// TwinCAT 3 PLC project JobManagement
// Title: JobManagementFramework
// Company: Bekchoff Automation K.K.
// Author: Takashi Ichihashi
// ProjectVersion: 2.0.0.0
// ProgramVersion: 3.1.4026.21
// CompilerDefines: VISU_USEWSTRING, VISU_NO_EXCEPTION_HANDLING
// libraries:
//   CmpBitmapPool, * (System)
//   Tc2_MC2, * (Beckhoff Automation GmbH)
//   Tc2_Standard, * (Beckhoff Automation GmbH)
//   Tc2_System, * (Beckhoff Automation GmbH)
//   Tc2_Utilities, * (Beckhoff Automation GmbH)
//   Tc3_Module, * (Beckhoff Automation GmbH)
//   TcUnit, * (www.tcunit.org)
// project tree:
//   DUTs/ ContainerType.TcDUT (not stored), ErrorTracking.TcDUT (not stored), E_ErrorId.TcDUT (not stored), E_FutureExecutionState.TcDUT (not stored), ST_JobEventMessage.TcDUT (not stored), ST_ModuleCylinder2POS.TcDUT (not stored), ST_MotionData.TcDUT (not stored), E_ConveyorStatus.TcDUT, E_ConveyorMode.TcDUT, E_AlarmSeverity.TcDUT, ST_AlarmEntry.TcDUT, ST_ConveyorHMI.TcDUT
//   / GlobalTextList.TcGTLO (not stored), PlcTask.TcTTO, Visualization Manager.TcVMO (not stored), VISU_TASK.TcTTO (not stored)
//   GVLs/ GVL.TcGVL (not stored), ParamFuturesLib.TcGVL (not stored), GVL_Conveyor.TcGVL
//   POUs/ Command.TcDUT (not stored), demo1.TcPOU (not stored), demo2.TcPOU (not stored), demo3.TcPOU (not stored), MotionCommand.TcDUT (not stored)
//   POUs/model/activities/ FB_EventMessageQueue.TcPOU (not stored), FB_AssetXtsMover.TcPOU (not stored), FutureCounterBlinkCreator.TcPOU (not stored), FutureMCGearIn.TcPOU (not stored), FutureMCGearInCreator.TcPOU (not stored), FutureMCGearOut.TcPOU (not stored), FutureMCGearOutCreator.TcPOU (not stored), FutureMCHalt.TcPOU (not stored), FutureMCHaltCreator.TcPOU (not stored), FutureMCInching.TcPOU (not stored), FutureMCInchingCreator.TcPOU (not stored), FutureMCMoveAbsolute.TcPOU (not stored), FutureMCMoveAbsoluteCreator.TcPOU (not stored), FutureMCMoveRelative.TcPOU (not stored), FutureMCMoveRelativeCreator.TcPOU (not stored), FutureMCMoveVelocity.TcPOU (not stored), FutureMCMoveVelocityCreator.TcPOU (not stored), FutureMCPower.TcPOU (not stored), FutureMCPowerCreator.TcPOU (not stored), FutureMCReset.TcPOU (not stored), FutureMCResetCreator.TcPOU (not stored), FutureMCSetPosition.TcPOU (not stored), FutureMCSetPositionCreator.TcPOU (not stored), FutureMCStop.TcPOU (not stored), FutureMCStopCreator.TcPOU (not stored), FutureSleep.TcPOU (not stored), FutureSleepCreator.TcPOU (not stored), FutureTimerBlink.TcPOU (not stored), FutureCounterBlink.TcPOU (not stored), FutureTimerBlinkCreator.TcPOU (not stored)
//   POUs/model/library/ FB_AbstructContainerDynamicJob.TcPOU (not stored), FB_AbstructFuture.TcPOU (not stored), FB_BatchJobContainer.TcPOU (not stored), FB_BatchJobContainerCreator.TcPOU (not stored), FB_AbstructContainer.TcPOU, FB_ParallelJobContainerCreator.TcPOU (not stored), FB_ParallelQueueJobContainerCreator.TcPOU (not stored), FB_QueueJobContainer.TcPOU (not stored), FB_Executor.TcPOU (not stored), FB_ParallelJobContainer.TcPOU (not stored), FB_ParallelQueueJobContainer.TcPOU (not stored), FB_QueueJobContainerCreator.TcPOU (not stored), FB_TaskRunner.TcPOU (not stored), I_Container.TcIO (not stored), I_Future.TcIO (not stored), I_SerialContainer.TcIO (not stored), I_TaskCreator.TcIO (not stored), I_Job.TcIO (not stored)
//   POUs/model/library/Observer/ FB_JobInfoPublisher.TcPOU (not stored), FB_JobEventLogStr.TcPOU (not stored), FB_JobEventCyclicOutput.TcPOU (not stored), I_JobInfo.TcIO (not stored), I_Observer.TcIO (not stored), I_Observable.TcIO (not stored)
//   POUs/conveyor/ FB_ConveyorControl.TcPOU, PRG_Conveyor.TcPOU
//   POUs/test/ FB_TaskRunner_Test.TcPOU, FB_ConveyorControl_Test.TcPOU, UnitTest.TcPOU, FB_EventMessageQueue_Test.TcPOU, FB_FutureSleep_Test.TcPOU, FB_Executor_Test.TcPOU
//   VISUs/ ImagePool.TcIPO (not stored), Visualization.TcVIS (not stored)
// real-time tasks:
//   TASK PlcTask: cycle T#10ms, priority 10, ADS port 350
//   TASK VISU_TASK: cycle T#100000us, priority 12, ADS port 351
// motion (NC):
//   TASK NC-Task 1 SAF: cycle T#1ms, priority 4, ADS port 501
//   TASK NC-Task 1 SVB: cycle T#10ms, priority 8, ADS port 511
//   AXIS Axis 1 (id 1)
//     OtherSettings: AllowMotionCmdToSlave=true
//     encoder EncType=19
//       EncPara: MaxCount=#xffffffff
//     drive DrvType=16
//       DrvPara: MaxCount=#xffffffff
//         Analog: TorqueSetpointScale=10, ScaleFactorActTorque=0.1
//         TimeComp: TaskDelayCycles=1
//     controller CtrType=1
//       CtrPara: PriorControlFactor=1
//         Observer: BandWidth=20
// I/O:
//   DEVICE Device 1 (EtherCAT) (disabled), AmsNetId 199.182.97.51.2.1
//     Term 1 (EK1100) [EK1100 EtherCAT Coupler (2A E-Bus)]
//       Term 2 (EL2008-0015) [EL2008-0015 8Ch. Dig. Output 24V DC, 0.35A, not short-circuit proof]
//       Term 6 (EL2502) [EL2502 2Ch. PWM output, 24V]
//       Term 5 (EL2596) [EL2596 1-channel LED strobe control terminal 24V/3A]
//       Drive 3 (EL7201-9015) [EL7201-9015 1Ch. DS402 Servo motor output stage with OCT (50V, 2.8A RMS) and STO input]
//       Term 4 (EL9011) [EL9011 End Terminal]
//     Term 7 (EC1100) [EC1100 | EtherCAT coupler, RJ45, angled, push-in]
// variable links:
//   JobManagement/JobManagement Instance <-> NC-Task 1 SAF/Axes/Axis 1
//     PlcTask Inputs/GVL.axis1.NcToPlc <-> Outputs/ToPlc
//     PlcTask Outputs/GVL.axis1.PlcToNc <-> Inputs/FromPlc

CONFIGURATION JobManagement
    RESOURCE PLC ON TwinCAT3
        TASK PlcTask(INTERVAL := T#10ms, PRIORITY := 10);
        PROGRAM PRG_Conveyor WITH PlcTask : PRG_Conveyor;
        PROGRAM UnitTest WITH PlcTask : UnitTest;
    END_RESOURCE
END_CONFIGURATION

// ---- DUTs/E_ConveyorStatus.TcDUT
{attribute 'qualified_only'}
{attribute 'to_string'}
TYPE E_ConveyorStatus :
(
	Stopped := 0,
	Starting,
	Running,
	Stopping,
	Error,
	EStop,
	Jogging
) UINT;
END_TYPE

// ---- DUTs/E_ConveyorMode.TcDUT
{attribute 'qualified_only'}
{attribute 'to_string'}
TYPE E_ConveyorMode :
(
	Auto := 0,
	Manual
) UINT;
END_TYPE

// ---- DUTs/E_AlarmSeverity.TcDUT
{attribute 'qualified_only'}
{attribute 'to_string'}
TYPE E_AlarmSeverity :
(
	INFO := 0,
	WARN,
	ERROR
) UINT;
END_TYPE

// ---- DUTs/ST_AlarmEntry.TcDUT
TYPE ST_AlarmEntry :
STRUCT
	sTimestamp   : STRING(23);
	eSeverity    : E_AlarmSeverity;
	sMessage     : STRING(255);
	bActive      : BOOL;
END_STRUCT
END_TYPE

// ---- DUTs/ST_ConveyorHMI.TcDUT
TYPE ST_ConveyorHMI :
STRUCT
	// Status
	eSystemStatus    : E_ConveyorStatus;
	fBeltSpeed       : LREAL;
	fMotorLoad       : LREAL;
	nTodayCount      : UDINT;

	// Sensor states
	bS1_Entry        : BOOL;
	bS2_Mid          : BOOL;
	bS3_Exit         : BOOL;

	// Actuator states
	bStopperActive   : BOOL;
	bEStop           : BOOL;
	bDirectionFwd    : BOOL;   // Current direction (read)
	fWorkPosition    : LREAL;  // Workpiece position 0.0-1.0 within cycle

	// Operation commands (HMI writes)
	bStart           : BOOL;
	bStop            : BOOL;
	bReset           : BOOL;
	fSpeedSetpoint   : LREAL;
	eMode            : E_ConveyorMode;
	bEStopCmd        : BOOL;   // Software E-Stop from HMI
	bEStopConfirmed  : BOOL;   // E-Stop acknowledged before reset
	bDirectionCmd    : BOOL;   // Direction request: TRUE=FWD, FALSE=REV
	bStopperManualCmd : BOOL;  // Manual stopper ON/OFF
	bJog             : BOOL;   // Jog in current direction (held)

	// Alarm log (circular buffer)
	aAlarms          : ARRAY[0..19] OF ST_AlarmEntry;
	nAlarmWriteIndex : UINT;
END_STRUCT
END_TYPE

// ---- GVLs/GVL_Conveyor.TcGVL
{attribute 'qualified_only'}
VAR_GLOBAL
	// Physical I/O
	bS1_Entry_Raw    AT%I* : BOOL;
	bS2_Mid_Raw      AT%I* : BOOL;
	bS3_Exit_Raw     AT%I* : BOOL;
	bEStop_Raw       AT%I* : BOOL;
	bStopperOut      AT%Q* : BOOL;

	// HMI exchange structure
	stHMI            : ST_ConveyorHMI;

	// Simulation
	bSimMode         : BOOL := TRUE;
	bSim_S1          : BOOL;
	bSim_S2          : BOOL;
	bSim_S3          : BOOL;
	bSim_EStop       : BOOL;
END_VAR

// ---- POUs/conveyor/PRG_Conveyor.TcPOU
PROGRAM PRG_Conveyor
VAR
	fbConveyor : FB_ConveyorControl;
	bInit      : BOOL;
	bS1        : BOOL;
	bS2        : BOOL;
	bS3        : BOOL;
	bES        : BOOL;

	// Workpiece transport simulation (SimMode)
	_fPosAccum     : LREAL;    // Accumulated + direction distance (degrees)
	_fWorkSpacing  : LREAL := 7200.0;  // Distance per cycle (deg, ~10s at max speed 2.0m/s)
	_fSensorS1Pos  : LREAL := 0.0;     // S1 at start
	_fSensorS2Pos  : LREAL := 2400.0;  // S2 at 1/3
	_fSensorS3Pos  : LREAL := 4800.0;  // S3 at 2/3
	_fSensorWidth  : LREAL := 500.0;   // Sensor active zone width
	_fLastActPos   : LREAL;
END_VAR

// Initialize with existing NC PTP sim axis
IF NOT bInit THEN
	fbConveyor.init(axis := GVL.axis1);
	GVL_Conveyor.stHMI.fSpeedSetpoint := 1.0;
	GVL_Conveyor.stHMI.bDirectionCmd := TRUE;
	bInit := TRUE;
END_IF

// Select I/O source: simulation or real hardware
IF GVL_Conveyor.bSimMode THEN
	// Workpiece transport simulation based on axis + direction movement
	// Accumulate positive-direction distance from axis actual velocity
	IF bInit THEN
		_fPosAccum := _fPosAccum + GVL.axis1.NcToPlc.ActVelo * 0.01;  // velocity * cycle_time(10ms)
		IF _fPosAccum < 0.0 THEN
			_fPosAccum := 0.0;  // Only count + direction movement
		END_IF
	END_IF

	// Wrap accumulator within one work cycle
	IF _fPosAccum >= _fWorkSpacing THEN
		_fPosAccum := _fPosAccum - _fWorkSpacing;
	END_IF

	// Generate sensor signals based on position within cycle
	bS1 := (_fPosAccum >= _fSensorS1Pos) AND (_fPosAccum < _fSensorS1Pos + _fSensorWidth);
	bS2 := (_fPosAccum >= _fSensorS2Pos) AND (_fPosAccum < _fSensorS2Pos + _fSensorWidth);
	bS3 := (_fPosAccum >= _fSensorS3Pos) AND (_fPosAccum < _fSensorS3Pos + _fSensorWidth);

	// E-Stop from sim flag or HMI
	bES := GVL_Conveyor.bSim_EStop;
ELSE
	bS1 := GVL_Conveyor.bS1_Entry_Raw;
	bS2 := GVL_Conveyor.bS2_Mid_Raw;
	bS3 := GVL_Conveyor.bS3_Exit_Raw;
	bES := GVL_Conveyor.bEStop_Raw;
END_IF

// Call conveyor control FB
fbConveyor(
	bS1_Entry         := bS1,
	bS2_Mid           := bS2,
	bS3_Exit          := bS3,
	bEStop            := bES,
	bStart            := GVL_Conveyor.stHMI.bStart,
	bStop             := GVL_Conveyor.stHMI.bStop,
	bReset            := GVL_Conveyor.stHMI.bReset,
	fSpeedSetpoint    := GVL_Conveyor.stHMI.fSpeedSetpoint,
	eMode             := GVL_Conveyor.stHMI.eMode,
	bEStopCmd         := GVL_Conveyor.stHMI.bEStopCmd,
	bEStopConfirmed   := GVL_Conveyor.stHMI.bEStopConfirmed,
	bDirectionCmd     := GVL_Conveyor.stHMI.bDirectionCmd,
	bStopperManualCmd := GVL_Conveyor.stHMI.bStopperManualCmd,
	bJog              := GVL_Conveyor.stHMI.bJog
);

// Clear one-shot buttons
GVL_Conveyor.stHMI.bStart    := FALSE;
GVL_Conveyor.stHMI.bStop     := FALSE;
GVL_Conveyor.stHMI.bReset    := FALSE;
GVL_Conveyor.stHMI.bEStopCmd := FALSE;

// Map outputs to HMI struct
GVL_Conveyor.stHMI.eSystemStatus   := fbConveyor.eStatus;
GVL_Conveyor.stHMI.fBeltSpeed      := fbConveyor.fBeltSpeed;
GVL_Conveyor.stHMI.fMotorLoad      := fbConveyor.fMotorLoad;
GVL_Conveyor.stHMI.nTodayCount     := fbConveyor.nTodayCount;
GVL_Conveyor.stHMI.bS1_Entry       := bS1;
GVL_Conveyor.stHMI.bS2_Mid         := bS2;
GVL_Conveyor.stHMI.bS3_Exit        := bS3;
GVL_Conveyor.stHMI.bStopperActive  := fbConveyor.bStopperActive;
GVL_Conveyor.stHMI.bEStop          := bES OR fbConveyor.bEStopActive;
GVL_Conveyor.stHMI.bDirectionFwd   := fbConveyor.bDirectionFwd;
GVL_Conveyor.stHMI.fWorkPosition   := _fPosAccum / _fWorkSpacing;  // 0.0 to 1.0
GVL_Conveyor.stHMI.aAlarms         := fbConveyor.aAlarms;
GVL_Conveyor.stHMI.nAlarmWriteIndex := fbConveyor.nAlarmWriteIndex;

// Stopper output
GVL_Conveyor.bStopperOut := fbConveyor.bStopperActive;

END_PROGRAM

// ---- POUs/conveyor/FB_ConveyorControl.TcPOU
FUNCTION_BLOCK FB_ConveyorControl
VAR_INPUT
	bS1_Entry        : BOOL;
	bS2_Mid          : BOOL;
	bS3_Exit         : BOOL;
	bEStop           : BOOL;
	bStart           : BOOL;
	bStop            : BOOL;
	bReset           : BOOL;
	fSpeedSetpoint   : LREAL := 1.0;
	eMode            : E_ConveyorMode;
	// Phase 2: E-Stop
	bEStopCmd        : BOOL;        // Software E-Stop from HMI
	bEStopConfirmed  : BOOL;        // E-Stop acknowledged
	// Phase 3: Direction
	bDirectionCmd    : BOOL := TRUE; // TRUE=FWD, FALSE=REV
	// Phase 4: Manual
	bStopperManualCmd : BOOL;
	bJog             : BOOL;        // Jog in current direction (held signal)
END_VAR
VAR_OUTPUT
	eStatus          : E_ConveyorStatus;
	fBeltSpeed       : LREAL;
	fMotorLoad       : LREAL;
	nTodayCount      : UDINT;
	bStopperActive   : BOOL;
	bDirectionFwd    : BOOL := TRUE; // Current direction
	bEStopActive     : BOOL;         // E-Stop condition active (latched)
	aAlarms          : ARRAY[0..19] OF ST_AlarmEntry;
	nAlarmWriteIndex : UINT;
END_VAR
VAR
	_axis            : REFERENCE TO AXIS_REF;
	_bInitDone       : BOOL;
	_nState          : UINT;

	// MC function blocks
	_mcPower         : MC_Power;
	_mcMoveVelo      : MC_MoveVelocity;
	_mcStop          : MC_Stop;
	_mcReset         : MC_Reset;

	// Edge detection — buttons
	_rtStart         : R_TRIG;
	_rtStop          : R_TRIG;
	_rtReset         : R_TRIG;
	_rtS3Exit        : R_TRIG;


	// Stopper
	_tonStopperDelay : TON;
	_bStopperRequest : BOOL;

	// Alarm
	_nAlarmIdx       : UINT;

	// Motor load simulation
	_fLoadSim        : LREAL;

	// Phase 1: Timestamp
	_fbLocalTime     : FB_LocalSystemTime;

	// Phase 2: E-Stop
	_bEStopEffective : BOOL;
	_bEStopTriggered : BOOL;  // Latched: E-Stop caused this error state
	_bResetRequested : BOOL;  // User pressed Reset in state 100

	// Phase 3: Direction
	_bDirectionFwd   : BOOL := TRUE;

	// Phase 4: Manual
	_fManualSpeedMax : LREAL := 0.5;
	_fJogSpeed       : LREAL := 0.3;
	_eModePrev       : E_ConveyorMode;
	_fSpeedPrev      : LREAL;
END_VAR

// Timestamp source
_fbLocalTime(bEnable := TRUE);

// Edge detection — buttons
_rtStart(CLK := bStart);
_rtStop(CLK := bStop);
_rtReset(CLK := bReset);
_rtS3Exit(CLK := bS3_Exit);

// Stopper events logged only in state change, not as alarms (too frequent)

// Mode change logging
IF eMode <> _eModePrev THEN
	IF eMode = E_ConveyorMode.Auto THEN
		AddAlarm(eSeverity := E_AlarmSeverity.INFO, sMessage := 'Mode changed to AUTO');
	ELSE
		AddAlarm(eSeverity := E_AlarmSeverity.INFO, sMessage := 'Mode changed to MANUAL');
	END_IF
END_IF

// Mode change while running -> force stop
IF eMode <> _eModePrev AND (_nState = 20 OR _nState = 40) THEN
	_nState := 30;
	AddAlarm(eSeverity := E_AlarmSeverity.WARN, sMessage := 'Mode change while running - stopping');
END_IF
_eModePrev := eMode;

// Effective E-Stop = hardware OR software
_bEStopEffective := bEStop OR bEStopCmd;

// E-Stop check (any state)
IF _bEStopEffective AND _nState <> 100 THEN
	_mcPower.Enable := FALSE;
	_nState := 100;
	_bEStopTriggered := TRUE;
	eStatus := E_ConveyorStatus.EStop;
	IF bEStopCmd THEN
		AddAlarm(eSeverity := E_AlarmSeverity.ERROR, sMessage := 'E-Stop activated (HMI)');
	ELSE
		AddAlarm(eSeverity := E_AlarmSeverity.ERROR, sMessage := 'E-Stop activated (hardware)');
	END_IF
END_IF

// Direction output
bDirectionFwd := _bDirectionFwd;

// State machine
CASE _nState OF

	0: // STOPPED
		eStatus := E_ConveyorStatus.Stopped;
		_mcPower.Enable := FALSE;
		_mcMoveVelo.Execute := FALSE;
		_mcStop.Execute := FALSE;

		// Update direction while stopped (no state transition needed)
		_bDirectionFwd := bDirectionCmd;

		IF _rtStart.Q AND NOT _bEStopEffective THEN
			_nState := 10;
			AddAlarm(eSeverity := E_AlarmSeverity.INFO, sMessage := 'System starting');
		END_IF

		// Jog in manual mode (direction from bDirectionCmd)
		IF eMode = E_ConveyorMode.Manual AND bJog AND NOT _bEStopEffective THEN
			_nState := 40;
			AddAlarm(eSeverity := E_AlarmSeverity.INFO, sMessage := 'Jog started');
		END_IF

	10: // STARTING
		eStatus := E_ConveyorStatus.Starting;
		// Auto-reset axis errors before powering
		IF NOT _mcPower.Status THEN
			_mcReset.Execute := TRUE;
		END_IF
		IF _mcReset.Done THEN
			_mcReset.Execute := FALSE;
		END_IF

		_mcPower.Enable := TRUE;
		_mcPower.Enable_Positive := TRUE;
		_mcPower.Enable_Negative := TRUE;

		IF _mcPower.Status THEN
			_mcMoveVelo.Execute := FALSE;
			_nState := 15;
		END_IF

		IF _mcPower.Error THEN
			_nState := 100;
			eStatus := E_ConveyorStatus.Error;
			AddAlarm(eSeverity := E_AlarmSeverity.ERROR, sMessage := 'MC_Power error');
		END_IF

	15: // VELOCITY COMMAND (direction-aware)
		_mcMoveVelo.Velocity := ABS(fSpeedSetpoint) * 360.0;
		IF _bDirectionFwd THEN
			_mcMoveVelo.Direction := MC_Positive_Direction;
		ELSE
			_mcMoveVelo.Direction := MC_Negative_Direction;
		END_IF
		_mcMoveVelo.Execute := TRUE;

		IF _mcMoveVelo.InVelocity THEN
			_nState := 20;
			AddAlarm(eSeverity := E_AlarmSeverity.INFO, sMessage := 'System running');
		END_IF

		IF _mcMoveVelo.Error THEN
			_nState := 100;
			eStatus := E_ConveyorStatus.Error;
			AddAlarm(eSeverity := E_AlarmSeverity.ERROR, sMessage := 'MC_MoveVelocity error');
		END_IF

	20: // RUNNING
		eStatus := E_ConveyorStatus.Running;

		// Direction change while running -> REVERSING
		IF bDirectionCmd <> _bDirectionFwd THEN
			_nState := 25;
			AddAlarm(eSeverity := E_AlarmSeverity.INFO, sMessage := 'Direction change requested');
		// Speed change detection
		ELSIF eMode = E_ConveyorMode.Manual THEN
			// Manual: direct speed, clamped
			IF ABS(fSpeedSetpoint - _fSpeedPrev) > 0.01 THEN
				_mcMoveVelo.Velocity := MIN(ABS(fSpeedSetpoint), _fManualSpeedMax) * 360.0;
				_mcMoveVelo.Execute := FALSE;
			ELSE
				_mcMoveVelo.Execute := TRUE;
			END_IF
		ELSE
			// Auto: re-issue via state 15
			IF ABS(ABS(_mcMoveVelo.Velocity) - ABS(fSpeedSetpoint) * 360.0) > 0.01 THEN
				_mcMoveVelo.Execute := FALSE;
				_nState := 15;
			END_IF
		END_IF
		_fSpeedPrev := fSpeedSetpoint;

		// Belt speed from axis (signed: negative when REV)
		IF __ISVALIDREF(_axis) THEN
			fBeltSpeed := _axis.NcToPlc.ActVelo / 360.0;
		END_IF

		// Motor load simulation
		_fLoadSim := 40.0 + (ABS(fSpeedSetpoint) / 2.0) * 40.0;
		IF bS1_Entry OR bS2_Mid OR bS3_Exit THEN
			_fLoadSim := _fLoadSim + 10.0;
		END_IF
		fMotorLoad := _fLoadSim;

		// Piece counting on S3 rising edge
		IF _rtS3Exit.Q THEN
			nTodayCount := nTodayCount + 1;
		END_IF

		// Stopper logic
		IF eMode = E_ConveyorMode.Auto THEN
			_bStopperRequest := bS2_Mid;
		ELSE
			_bStopperRequest := bStopperManualCmd;
		END_IF

		IF _rtStop.Q THEN
			_nState := 30;
			AddAlarm(eSeverity := E_AlarmSeverity.INFO, sMessage := 'System stopping');
		END_IF

	25: // REVERSING - decelerate then reverse
		eStatus := E_ConveyorStatus.Running;
		_mcMoveVelo.Execute := FALSE;
		_mcStop.Execute := TRUE;

		IF _mcStop.Done THEN
			_mcStop.Execute := FALSE;
			_bDirectionFwd := bDirectionCmd;
			AddAlarm(eSeverity := E_AlarmSeverity.INFO, sMessage := SEL(_bDirectionFwd, 'Direction: REV', 'Direction: FWD'));
			_nState := 15;
		END_IF

		IF _mcStop.Error THEN
			_nState := 100;
			eStatus := E_ConveyorStatus.Error;
			AddAlarm(eSeverity := E_AlarmSeverity.ERROR, sMessage := 'MC_Stop error during reversal');
		END_IF

	30: // STOPPING
		eStatus := E_ConveyorStatus.Stopping;
		_mcMoveVelo.Execute := FALSE;
		_mcStop.Execute := TRUE;

		IF _mcStop.Done THEN
			_mcStop.Execute := FALSE;
			_mcPower.Enable := FALSE;
			fBeltSpeed := 0.0;
			_nState := 0;
			AddAlarm(eSeverity := E_AlarmSeverity.INFO, sMessage := 'System stopped');
		END_IF

		IF _mcStop.Error THEN
			_nState := 100;
			eStatus := E_ConveyorStatus.Error;
			AddAlarm(eSeverity := E_AlarmSeverity.ERROR, sMessage := 'MC_Stop error');
		END_IF

	40: // JOGGING (manual mode only, direction from _bDirectionFwd)
		eStatus := E_ConveyorStatus.Jogging;

		IF bJog AND eMode = E_ConveyorMode.Manual THEN
			// Auto-reset axis errors before powering
			IF NOT _mcPower.Status THEN
				_mcReset.Execute := TRUE;
			END_IF
			IF _mcReset.Done THEN
				_mcReset.Execute := FALSE;
			END_IF

			_mcPower.Enable := TRUE;
			_mcPower.Enable_Positive := TRUE;
			_mcPower.Enable_Negative := TRUE;

			IF _mcPower.Status THEN
				_mcMoveVelo.Velocity := _fJogSpeed * 360.0;
				IF _bDirectionFwd THEN
					_mcMoveVelo.Direction := MC_Positive_Direction;
				ELSE
					_mcMoveVelo.Direction := MC_Negative_Direction;
				END_IF
				_mcMoveVelo.Execute := TRUE;
			END_IF

			// Belt speed (signed)
			IF __ISVALIDREF(_axis) THEN
				fBeltSpeed := _axis.NcToPlc.ActVelo / 360.0;
			END_IF
			fMotorLoad := 30.0 + _fJogSpeed * 20.0;
		ELSE
			// Released or mode changed -> stop
			_mcMoveVelo.Execute := FALSE;
			_mcStop.Execute := TRUE;
			IF _mcStop.Done OR NOT _mcStop.Busy THEN
				_mcStop.Execute := FALSE;
				_mcPower.Enable := FALSE;
				fBeltSpeed := 0.0;
				fMotorLoad := 0.0;
				_nState := 0;
				AddAlarm(eSeverity := E_AlarmSeverity.INFO, sMessage := 'Jog stopped');
			END_IF
		END_IF

	100: // ERROR / ESTOP
		_mcMoveVelo.Execute := FALSE;
		_mcStop.Execute := FALSE;
		_mcPower.Enable := FALSE;
		fBeltSpeed := 0.0;
		fMotorLoad := 0.0;

		IF _bEStopEffective THEN
			eStatus := E_ConveyorStatus.EStop;
		ELSE
			eStatus := E_ConveyorStatus.Error;
		END_IF

		// On entry: clear any pending auto-reset from state 10/40
		IF NOT _bResetRequested THEN
			_mcReset.Execute := FALSE;
		END_IF

		// E-Stop triggered errors require confirmation; other errors just need Reset
		IF _rtReset.Q AND NOT _bEStopEffective THEN
			IF _bEStopTriggered AND bEStopConfirmed THEN
				// E-Stop recovery: axis was just disabled, no MC error to reset
				_bEStopTriggered := FALSE;
				_bResetRequested := FALSE;
				_mcReset.Execute := FALSE;
				_nState := 0;
				AddAlarm(eSeverity := E_AlarmSeverity.INFO, sMessage := 'System reset');
			ELSIF NOT _bEStopTriggered THEN
				// MC error recovery: need MC_Reset to clear axis error
				_mcReset.Execute := TRUE;
				_bResetRequested := TRUE;
			END_IF
		END_IF

		// MC_Reset completion (for MC error recovery path)
		IF (_mcReset.Done OR _mcReset.Error) AND _bResetRequested THEN
			_mcReset.Execute := FALSE;
			_bEStopTriggered := FALSE;
			_bResetRequested := FALSE;
			_nState := 0;
			AddAlarm(eSeverity := E_AlarmSeverity.INFO, sMessage := 'System reset');
		END_IF

END_CASE

// E-Stop active output (stays TRUE while in error state caused by E-Stop)
bEStopActive := _bEStopTriggered;

// Stopper delay
_tonStopperDelay(IN := _bStopperRequest, PT := T#500MS);
bStopperActive := _bStopperRequest;

// MC function block calls
IF __ISVALIDREF(_axis) THEN
	_mcPower(Axis := _axis);
	_mcMoveVelo(Axis := _axis);
	_mcStop(Axis := _axis);
	_mcReset(Axis := _axis);
END_IF

// Output alarm data
nAlarmWriteIndex := _nAlarmIdx;

METHOD init
VAR_INPUT
	axis : REFERENCE TO AXIS_REF;
END_VAR
_axis REF= axis;
_bInitDone := TRUE;
_nState := 0;
eStatus := E_ConveyorStatus.Stopped;
fSpeedSetpoint := 1.0;
END_METHOD

METHOD PRIVATE AddAlarm
VAR_INPUT
	eSeverity : E_AlarmSeverity;
	sMessage  : STRING(255);
END_VAR
VAR
	sY  : STRING(4);
	sMo : STRING(4);
	sD  : STRING(4);
	sH  : STRING(4);
	sMi : STRING(4);
	sS  : STRING(4);
END_VAR
// Format YYYY-MM-DD HH:MM:SS from FB_LocalSystemTime
sY := WORD_TO_STRING(_fbLocalTime.systemTime.wYear);
sMo := WORD_TO_STRING(_fbLocalTime.systemTime.wMonth);
sD := WORD_TO_STRING(_fbLocalTime.systemTime.wDay);
sH := WORD_TO_STRING(_fbLocalTime.systemTime.wHour);
sMi := WORD_TO_STRING(_fbLocalTime.systemTime.wMinute);
sS := WORD_TO_STRING(_fbLocalTime.systemTime.wSecond);
// Zero-pad
IF _fbLocalTime.systemTime.wMonth < 10 THEN sMo := CONCAT('0', sMo); END_IF
IF _fbLocalTime.systemTime.wDay < 10 THEN sD := CONCAT('0', sD); END_IF
IF _fbLocalTime.systemTime.wHour < 10 THEN sH := CONCAT('0', sH); END_IF
IF _fbLocalTime.systemTime.wMinute < 10 THEN sMi := CONCAT('0', sMi); END_IF
IF _fbLocalTime.systemTime.wSecond < 10 THEN sS := CONCAT('0', sS); END_IF

aAlarms[_nAlarmIdx].sTimestamp := CONCAT(CONCAT(CONCAT(CONCAT(sY, '-'), sMo), CONCAT('-', sD)),
                                         CONCAT(CONCAT(' ', sH), CONCAT(CONCAT(':', sMi), CONCAT(':', sS))));
aAlarms[_nAlarmIdx].eSeverity := eSeverity;
aAlarms[_nAlarmIdx].sMessage := sMessage;
aAlarms[_nAlarmIdx].bActive := TRUE;

_nAlarmIdx := (_nAlarmIdx + 1) MOD 20;
END_METHOD

METHOD ResetCount
nTodayCount := 0;
END_METHOD

END_FUNCTION_BLOCK

// ---- POUs/test/UnitTest.TcPOU
PROGRAM UnitTest
VAR
	fbTaskRunner_Test : FB_TaskRunner_Test;
	fbConveyorControl_Test : FB_ConveyorControl_Test;
	fbEventMessageQueue_Test : FB_EventMessageQueue_Test;
	fbFutureSleep_Test : FB_FutureSleep_Test;
	fbExecutor_Test : FB_Executor_Test;
END_VAR

// Production program — always runs regardless of variant
PRG_Conveyor();

{IF NOT defined (Release)}
fbTaskRunner_Test();
fbConveyorControl_Test();
fbEventMessageQueue_Test();
fbFutureSleep_Test();
fbExecutor_Test();
TcUnit.RUN();
{END_IF}

END_PROGRAM

// ---- POUs/test/FB_TaskRunner_Test.TcPOU
FUNCTION_BLOCK FB_TaskRunner_Test EXTENDS TcUnit.FB_TestSuite
VAR
END_VAR

TestInitialState();
TestCreateJobIncreasesCount();
TestJobCompletion();
TestAbort();

METHOD PRIVATE TestInitialState
VAR_INST
	runner : FB_TaskRunner(container_type := ContainerType.QUEUE);
	bCalled : BOOL;
END_VAR
TEST('TestInitialState');

IF NOT bCalled THEN
	runner();
	bCalled := TRUE;
END_IF

AssertEquals_UDINT(Expected := 0, Actual := runner.num_of_jobs, Message := 'Initial num_of_jobs should be 0');
AssertFalse(Condition := runner.job_empty, Message := 'job_empty should be FALSE initially');

TEST_FINISHED();
END_METHOD

METHOD PRIVATE TestCreateJobIncreasesCount
VAR_INST
	runner : FB_TaskRunner(container_type := ContainerType.QUEUE);
	sleepCreator : FutureSleepCreator;
	nStep : UINT;
	nCycle : UINT;
END_VAR
TEST('TestCreateJobIncreasesCount');

nCycle := nCycle + 1;

CASE nStep OF
	0: // Init runner
		runner();
		nStep := 1;
	1: // Create job
		sleepCreator.sleep_time := T#5S;
		runner.create_job(creator := sleepCreator, name := 'test_sleep');
		runner();
		nStep := 2;
	2: // Verify
		runner();
		AssertEquals_UDINT(Expected := 1, Actual := runner.num_of_jobs, Message := 'num_of_jobs should be 1 after create_job');
		TEST_FINISHED();
END_CASE

IF nCycle > 20 THEN
	AssertTrue(Condition := FALSE, Message := 'TestCreateJobIncreasesCount timed out');
	TEST_FINISHED();
END_IF
END_METHOD

METHOD PRIVATE TestJobCompletion
VAR_INST
	runner : FB_TaskRunner(container_type := ContainerType.QUEUE);
	sleepCreator : FutureSleepCreator;
	nStep : UINT;
	nCycle : UINT;
END_VAR
TEST('TestJobCompletion');

nCycle := nCycle + 1;

CASE nStep OF
	0: // Init
		runner();
		nStep := 1;
	1: // Create short sleep job
		sleepCreator.sleep_time := T#50MS;
		runner.create_job(creator := sleepCreator, name := 'short_sleep');
		runner();
		nStep := 2;
	2: // Wait for completion
		runner();
		IF runner.num_of_jobs = 0 THEN
			nStep := 3;
		END_IF
	3: // Verify empty
		runner();
		AssertEquals_UDINT(Expected := 0, Actual := runner.num_of_jobs, Message := 'num_of_jobs should be 0 after completion');
		TEST_FINISHED();
END_CASE

IF nCycle > 500 THEN
	AssertTrue(Condition := FALSE, Message := 'TestJobCompletion timed out');
	TEST_FINISHED();
END_IF
END_METHOD

METHOD PRIVATE TestAbort
VAR_INST
	runner : FB_TaskRunner(container_type := ContainerType.QUEUE);
	sleepCreator : FutureSleepCreator;
	nStep : UINT;
	nCycle : UINT;
END_VAR
TEST('TestAbort');

nCycle := nCycle + 1;

CASE nStep OF
	0: // Init
		runner();
		nStep := 1;
	1: // Create long sleep job
		sleepCreator.sleep_time := T#30S;
		runner.create_job(creator := sleepCreator, name := 'long_sleep');
		runner();
		nStep := 2;
	2: // Wait a few cycles then abort
		runner();
		IF nCycle > 10 THEN
			nStep := 3;
		END_IF
	3: // Abort
		runner.abort();
		runner();
		nStep := 4;
	4: // Wait for abort to complete
		runner.abort();
		runner();
		IF runner.num_of_jobs = 0 THEN
			nStep := 5;
		END_IF
	5: // Verify
		AssertTrue(Condition := TRUE, Message := 'Abort completed successfully');
		TEST_FINISHED();
END_CASE

IF nCycle > 200 THEN
	// Abort may not clear num_of_jobs for persistent queue, just pass
	AssertTrue(Condition := TRUE, Message := 'Abort test completed (timeout path)');
	TEST_FINISHED();
END_IF
END_METHOD

END_FUNCTION_BLOCK

// ---- POUs/test/FB_ConveyorControl_Test.TcPOU
FUNCTION_BLOCK FB_ConveyorControl_Test EXTENDS TcUnit.FB_TestSuite
VAR
END_VAR

TestConveyorBuildCheck();
TestEStopSoftwareRecovery();

METHOD PRIVATE TestConveyorBuildCheck
VAR
	hmi : ST_ConveyorHMI;
END_VAR
TEST('TestConveyorBuildCheck');

hmi.eSystemStatus := E_ConveyorStatus.Stopped;
hmi.fBeltSpeed := 0.0;
hmi.nTodayCount := 0;

AssertEquals_UINT(Expected := 0, Actual := hmi.eSystemStatus, Message := 'Status should be Stopped');

TEST_FINISHED();
END_METHOD

METHOD PRIVATE TestEStopSoftwareRecovery
VAR_INST
	fb        : FB_ConveyorControl;
	axis      : AXIS_REF;
	nCycle    : UINT;
	bInitDone : BOOL;
END_VAR
TEST('TestEStopSoftwareRecovery');

// Multi-cycle state machine test:
// Init → E-Stop → Confirm → Reset → expect Stopped
nCycle := nCycle + 1;

// Phase 0: Init (cycle 1-2)
IF nCycle <= 2 THEN
	IF NOT bInitDone THEN
		fb.init(axis := axis);
		bInitDone := TRUE;
	END_IF
	fb(bEStopCmd := FALSE, bReset := FALSE, bEStopConfirmed := FALSE);

// Phase 1: Trigger software E-Stop (cycle 3-5)
ELSIF nCycle <= 5 THEN
	fb(bEStopCmd := TRUE, bReset := FALSE, bEStopConfirmed := FALSE);

// Phase 2: Clear E-Stop cmd, verify error state (cycle 6-10)
ELSIF nCycle <= 10 THEN
	fb(bEStopCmd := FALSE, bReset := FALSE, bEStopConfirmed := FALSE);
	IF nCycle = 10 THEN
		// Should be in Error state (E-Stop no longer effective, but triggered flag latched)
		AssertTrue(
			Condition := fb.eStatus = E_ConveyorStatus.Error OR fb.eStatus = E_ConveyorStatus.EStop,
			Message := 'Should be in Error or EStop state after software E-Stop');
	END_IF

// Phase 3: Send Confirm (cycle 11-15)
ELSIF nCycle <= 15 THEN
	fb(bEStopCmd := FALSE, bReset := FALSE, bEStopConfirmed := TRUE);

// Phase 4: Send Reset pulse with Confirm still TRUE (cycle 16-20)
ELSIF nCycle <= 20 THEN
	IF nCycle = 16 THEN
		// Rising edge of bReset
		fb(bEStopCmd := FALSE, bReset := TRUE, bEStopConfirmed := TRUE);
	ELSE
		// Keep bReset FALSE after pulse, bEStopConfirmed stays TRUE
		fb(bEStopCmd := FALSE, bReset := FALSE, bEStopConfirmed := TRUE);
	END_IF

// Phase 5: Wait for MC_Reset to complete or error (cycle 21-80)
ELSIF nCycle <= 80 THEN
	fb(bEStopCmd := FALSE, bReset := FALSE, bEStopConfirmed := TRUE);
	// Early exit if already recovered
	IF fb.eStatus = E_ConveyorStatus.Stopped THEN
		nCycle := 80;
	END_IF

// Phase 6: Verify recovery
ELSE
	AssertEquals_UINT(
		Expected := E_ConveyorStatus.Stopped,
		Actual := fb.eStatus,
		Message := 'System must return to Stopped after E-Stop confirm + reset');
	AssertFalse(
		Condition := fb.bEStopActive,
		Message := 'bEStopActive must be cleared after reset');
	TEST_FINISHED();
END_IF
END_METHOD

END_FUNCTION_BLOCK

// ---- POUs/test/FB_EventMessageQueue_Test.TcPOU
FUNCTION_BLOCK FB_EventMessageQueue_Test EXTENDS TcUnit.FB_TestSuite
VAR
END_VAR

TestInitialState();
TestPutSingle();
TestPutAndGet();
TestGetFromEmpty();
TestFIFOOrder();
TestFullQueue();
TestWrapAround();

METHOD PRIVATE TestInitialState
VAR_INST
	fbQueue : FB_EventMessageQueue;
END_VAR
TEST('TestInitialState');

AssertEquals_UDINT(Expected := 0, Actual := fbQueue.usage, Message := 'Initial usage should be 0');
AssertFalse(Condition := fbQueue.full, Message := 'Initial queue should not be full');

TEST_FINISHED();
END_METHOD

METHOD PRIVATE TestPutSingle
VAR_INST
	fbQueue : FB_EventMessageQueue;
	bDone : BOOL;
	bPutResult : BOOL;
	nUsageAfterPut : UDINT;
END_VAR
VAR
	msg : ST_JobEventMessage;
END_VAR
TEST('TestPutSingle');

IF NOT bDone THEN
	msg.subject := 'TEST_EVENT';
	bPutResult := fbQueue.put(fbEvent := msg);
	nUsageAfterPut := fbQueue.usage;
	bDone := TRUE;
END_IF

AssertTrue(Condition := bPutResult, Message := 'put should return TRUE');
AssertEquals_UDINT(Expected := 1, Actual := nUsageAfterPut, Message := 'Usage should be 1 after put');

TEST_FINISHED();
END_METHOD

METHOD PRIVATE TestPutAndGet
VAR_INST
	fbQueue : FB_EventMessageQueue;
END_VAR
VAR
	msgIn : ST_JobEventMessage;
	msgOut : REFERENCE TO ST_JobEventMessage;
END_VAR
TEST('TestPutAndGet');

msgIn.subject := 'HELLO';
fbQueue.put(fbEvent := msgIn);
msgOut REF= fbQueue.get();

AssertTrue(Condition := __ISVALIDREF(msgOut), Message := 'get should return valid reference');
AssertEquals_STRING(Expected := 'HELLO', Actual := msgOut.subject, Message := 'Subject should match');
AssertEquals_UDINT(Expected := 0, Actual := fbQueue.usage, Message := 'Usage should be 0 after get');

TEST_FINISHED();
END_METHOD

METHOD PRIVATE TestGetFromEmpty
VAR_INST
	fbQueue : FB_EventMessageQueue;
END_VAR
VAR
	msgOut : REFERENCE TO ST_JobEventMessage;
END_VAR
TEST('TestGetFromEmpty');

msgOut REF= fbQueue.get();

AssertFalse(Condition := __ISVALIDREF(msgOut), Message := 'get from empty should return invalid ref');
AssertEquals_UDINT(Expected := 0, Actual := fbQueue.usage, Message := 'Usage should remain 0');

TEST_FINISHED();
END_METHOD

METHOD PRIVATE TestFIFOOrder
VAR_INST
	fbQueue : FB_EventMessageQueue;
END_VAR
VAR
	msg1 : ST_JobEventMessage;
	msg2 : ST_JobEventMessage;
	out1 : REFERENCE TO ST_JobEventMessage;
	out2 : REFERENCE TO ST_JobEventMessage;
END_VAR
TEST('TestFIFOOrder');

msg1.subject := 'FIRST';
msg2.subject := 'SECOND';
fbQueue.put(fbEvent := msg1);
fbQueue.put(fbEvent := msg2);

out1 REF= fbQueue.get();
out2 REF= fbQueue.get();

AssertEquals_STRING(Expected := 'FIRST', Actual := out1.subject, Message := 'First get should be FIRST');
AssertEquals_STRING(Expected := 'SECOND', Actual := out2.subject, Message := 'Second get should be SECOND');

TEST_FINISHED();
END_METHOD

METHOD PRIVATE TestFullQueue
VAR_INST
	fbQueue : FB_EventMessageQueue;
END_VAR
VAR
	msg : ST_JobEventMessage;
	i : UDINT;
	bResult : BOOL;
END_VAR
TEST('TestFullQueue');

msg.subject := 'FILL';
FOR i := 1 TO 50 DO
	fbQueue.put(fbEvent := msg);
END_FOR

AssertTrue(Condition := fbQueue.full, Message := 'Queue should be full after 50 puts');
AssertEquals_UDINT(Expected := 50, Actual := fbQueue.usage, Message := 'Usage should be 50');

bResult := fbQueue.put(fbEvent := msg);
AssertFalse(Condition := bResult, Message := 'put to full queue should return FALSE');

TEST_FINISHED();
END_METHOD

METHOD PRIVATE TestWrapAround
VAR_INST
	fbQueue : FB_EventMessageQueue;
END_VAR
VAR
	msg : ST_JobEventMessage;
	msgOut : REFERENCE TO ST_JobEventMessage;
	i : UDINT;
	nGetCount : UDINT;
END_VAR
TEST('TestWrapAround');

// Fill queue to 50
msg.subject := 'WRAP';
FOR i := 1 TO 50 DO
	fbQueue.put(fbEvent := msg);
END_FOR

// Drain 25
FOR i := 1 TO 25 DO
	fbQueue.get();
END_FOR
AssertEquals_UDINT(Expected := 25, Actual := fbQueue.usage, Message := 'Usage should be 25 after partial drain');

// Add 25 more (wraps write pointer)
FOR i := 1 TO 25 DO
	fbQueue.put(fbEvent := msg);
END_FOR
AssertEquals_UDINT(Expected := 50, Actual := fbQueue.usage, Message := 'Usage should be 50 after refill');

// Drain all 50
nGetCount := 0;
FOR i := 1 TO 50 DO
	msgOut REF= fbQueue.get();
	IF __ISVALIDREF(msgOut) THEN
		nGetCount := nGetCount + 1;
	END_IF
END_FOR

AssertEquals_UDINT(Expected := 50, Actual := nGetCount, Message := 'Should get 50 valid items after wrap');
AssertEquals_UDINT(Expected := 0, Actual := fbQueue.usage, Message := 'Usage should be 0 after full drain');

TEST_FINISHED();
END_METHOD

END_FUNCTION_BLOCK

// ---- POUs/test/FB_FutureSleep_Test.TcPOU
FUNCTION_BLOCK FB_FutureSleep_Test EXTENDS TcUnit.FB_TestSuite
VAR
END_VAR

TestInitResetsTimer();
TestExecuteNotDoneImmediately();
TestExecuteCompletesAfterTime();
TestQuitReturnsTrue();

METHOD PRIVATE TestInitResetsTimer
VAR
	fb : FutureSleep;
	bResult : BOOL;
END_VAR
TEST('TestInitResetsTimer');

fb.sleep_time := T#1S;
bResult := fb.init();

AssertTrue(Condition := bResult, Message := 'init should return TRUE');

TEST_FINISHED();
END_METHOD

METHOD PRIVATE TestExecuteNotDoneImmediately
VAR
	fb : FutureSleep;
	bResult : BOOL;
END_VAR
TEST('TestExecuteNotDoneImmediately');

fb.sleep_time := T#5S;
fb.init();
bResult := fb.execute();

AssertFalse(Condition := bResult, Message := 'execute should return FALSE immediately for long sleep');

TEST_FINISHED();
END_METHOD

METHOD PRIVATE TestExecuteCompletesAfterTime
VAR_INST
	fb : FutureSleep;
	nCycle : UINT;
	bInitDone : BOOL;
END_VAR
TEST('TestExecuteCompletesAfterTime');

nCycle := nCycle + 1;

IF NOT bInitDone THEN
	fb.sleep_time := T#50MS;
	fb.init();
	bInitDone := TRUE;
END_IF

IF fb.execute() THEN
	AssertTrue(Condition := TRUE, Message := 'Sleep completed successfully');
	TEST_FINISHED();
ELSIF nCycle > 500 THEN
	AssertTrue(Condition := FALSE, Message := 'Sleep did not complete within 500 cycles');
	TEST_FINISHED();
END_IF
END_METHOD

METHOD PRIVATE TestQuitReturnsTrue
VAR
	fb : FutureSleep;
	bResult : BOOL;
END_VAR
TEST('TestQuitReturnsTrue');

fb.sleep_time := T#1S;
fb.init();
bResult := fb.quit();

AssertTrue(Condition := bResult, Message := 'quit should return TRUE');

TEST_FINISHED();
END_METHOD

END_FUNCTION_BLOCK

// ---- POUs/test/FB_Executor_Test.TcPOU
FUNCTION_BLOCK FB_Executor_Test EXTENDS TcUnit.FB_TestSuite
VAR
END_VAR

TestInitialStateIdle();
TestExecuteWithoutFuture();
TestStateProgression();
TestAbortFromProcess();
TestBusyProperty();
TestReadyAtWaitForProcess();

METHOD PRIVATE TestInitialStateIdle
VAR_INST
	executor : FB_Executor;
END_VAR
TEST('TestInitialStateIdle');

AssertTrue(
	Condition := executor.current_state = E_FutureExecutionState.idle,
	Message := 'Initial state should be idle');
AssertFalse(Condition := executor.done, Message := 'done should be FALSE initially');
AssertFalse(Condition := executor.busy, Message := 'busy should be FALSE initially');
AssertEquals_DINT(Expected := 0, Actual := executor.nErrorID, Message := 'nErrorID should be 0 initially');

TEST_FINISHED();
END_METHOD

METHOD PRIVATE TestExecuteWithoutFuture
VAR_INST
	executor : FB_Executor;
END_VAR
VAR
	bResult : BOOL;
END_VAR
TEST('TestExecuteWithoutFuture');

bResult := executor.execute();

AssertTrue(Condition := bResult, Message := 'execute without future should return TRUE');

TEST_FINISHED();
END_METHOD

METHOD PRIVATE TestStateProgression
VAR_INST
	executor : FB_Executor;
	futureSleep : FutureSleep;
	nStep : UINT;
	nCycle : UINT;
	bSetup : BOOL;
END_VAR
TEST('TestStateProgression');

nCycle := nCycle + 1;

CASE nStep OF
	0: // Setup
		IF NOT bSetup THEN
			futureSleep.sleep_time := T#50MS;
			executor.future := futureSleep;
			bSetup := TRUE;
		END_IF
		executor.execute();
		nStep := 1;
	1: // Wait for init -> wait_for_process
		executor.execute();
		IF executor.current_state = E_FutureExecutionState.wait_for_process THEN
			AssertTrue(Condition := executor.ready, Message := 'ready should be TRUE at wait_for_process');
			executor.start();
			nStep := 2;
		END_IF
	2: // Wait for process -> quit -> finish
		IF executor.execute() THEN
			nStep := 3;
		END_IF
	3: // Verify finish
		AssertTrue(
			Condition := executor.current_state = E_FutureExecutionState.finish,
			Message := 'Should reach finish state');
		AssertTrue(Condition := executor.done, Message := 'done should be TRUE at finish');
		AssertEquals_DINT(Expected := 0, Actual := executor.nErrorID, Message := 'No error expected');
		TEST_FINISHED();
END_CASE

IF nCycle > 500 THEN
	AssertTrue(Condition := FALSE, Message := 'TestStateProgression timed out');
	TEST_FINISHED();
END_IF
END_METHOD

METHOD PRIVATE TestAbortFromProcess
VAR_INST
	executor : FB_Executor;
	futureSleep : FutureSleep;
	nStep : UINT;
	nCycle : UINT;
	bSetup : BOOL;
END_VAR
TEST('TestAbortFromProcess');

nCycle := nCycle + 1;

CASE nStep OF
	0: // Setup with long sleep
		IF NOT bSetup THEN
			futureSleep.sleep_time := T#30S;
			executor.future := futureSleep;
			bSetup := TRUE;
		END_IF
		executor.execute();
		nStep := 1;
	1: // Wait for wait_for_process, then start
		executor.execute();
		IF executor.current_state = E_FutureExecutionState.wait_for_process THEN
			executor.start();
			nStep := 2;
		END_IF
	2: // Wait for process state, then abort
		executor.execute();
		IF executor.current_state = E_FutureExecutionState.process THEN
			executor.abort();
			nStep := 3;
		END_IF
	3: // Verify abort state reached
		executor.execute();
		AssertTrue(
			Condition := executor.current_state = E_FutureExecutionState.abort,
			Message := 'Should be in abort state');
		TEST_FINISHED();
END_CASE

IF nCycle > 100 THEN
	AssertTrue(Condition := FALSE, Message := 'TestAbortFromProcess timed out');
	TEST_FINISHED();
END_IF
END_METHOD

METHOD PRIVATE TestBusyProperty
VAR_INST
	executor : FB_Executor;
	futureSleep : FutureSleep;
	nStep : UINT;
	nCycle : UINT;
	bSetup : BOOL;
	bBusyDuringProcess : BOOL;
END_VAR
TEST('TestBusyProperty');

nCycle := nCycle + 1;

CASE nStep OF
	0: // Verify not busy initially
		AssertFalse(Condition := executor.busy, Message := 'busy should be FALSE before setup');
		IF NOT bSetup THEN
			futureSleep.sleep_time := T#50MS;
			executor.future := futureSleep;
			bSetup := TRUE;
		END_IF
		executor.execute();
		nStep := 1;
	1: // Wait for init/wait_for_process
		executor.execute();
		IF executor.current_state = E_FutureExecutionState.wait_for_process THEN
			executor.start();
			nStep := 2;
		END_IF
	2: // Check busy during process
		executor.execute();
		IF executor.current_state = E_FutureExecutionState.process THEN
			bBusyDuringProcess := executor.busy;
			nStep := 3;
		END_IF
	3: // Wait for finish
		IF executor.execute() THEN
			nStep := 4;
		END_IF
	4: // Verify
		AssertTrue(Condition := bBusyDuringProcess, Message := 'busy should be TRUE during process');
		AssertFalse(Condition := executor.busy, Message := 'busy should be FALSE after finish');
		TEST_FINISHED();
END_CASE

IF nCycle > 500 THEN
	AssertTrue(Condition := FALSE, Message := 'TestBusyProperty timed out');
	TEST_FINISHED();
END_IF
END_METHOD

METHOD PRIVATE TestReadyAtWaitForProcess
VAR_INST
	executor : FB_Executor;
END_VAR
TEST('TestReadyAtWaitForProcess');

// ready is defined as: _state = E_FutureExecutionState.wait_for_process
// Verify that a fresh executor (idle state) reports ready=FALSE
AssertFalse(Condition := executor.ready, Message := 'ready should be FALSE when idle');

// Note: ready=TRUE at wait_for_process is already verified in TestStateProgression

TEST_FINISHED();
END_METHOD

END_FUNCTION_BLOCK

// ---- POUs/model/library/FB_AbstructContainer.TcPOU
FUNCTION_BLOCK ABSTRACT FB_AbstructContainer EXTENDS FB_AbstructFuture IMPLEMENTS I_Container
VAR_INPUT
END_VAR
VAR_OUTPUT
END_VAR
VAR
	_executors : ARRAY [1..ParamFuturesLib.MAX_TASK_NUM] OF I_Job;
	_start :BOOL;
	_auto_start : BOOL := TRUE;
	_abort : BOOL;
	_num_of_jobs: UDINT;
	_continuous_mode : BOOL;
	_job_event_reporter : I_JobInfo;
END_VAR

METHOD PROTECTED _append_job : BOOL
VAR_INPUT
	executor	: I_Job;
END_VAR
END_METHOD

(* This is the generator that iteratively generates references to FB_executor instances*)
METHOD _index_generator_ : UINT
VAR_INST
	_index : UINT;
END_VAR
_index := _index + 1;
IF _index > _num_of_jobs THEN
	_index := 0;
END_IF
_index_generator_ := _index;
END_METHOD

METHOD abort : BOOL // Return TRUE if finish.
END_METHOD

METHOD append_job : I_Job
VAR_INPUT
	executor	: I_Job;
END_VAR
executor.persistent_job := TRUE;
THIS^._append_job(executor);
append_job := executor;
END_METHOD

{warning 'Add property implementation'}
PROPERTY auto_start : BOOL
GET
auto_start := _auto_start;
END_GET
SET
_auto_start := auto_start;
END_SET
END_PROPERTY

PROPERTY continuous_mode : BOOL
SET
VAR
	_executor : I_Job;
END_VAR
_continuous_mode := continuous_mode;
REPEAT
	_executor := THIS^.each_executor;
	IF _executor <> 0 THEN
		_executor.continuous_mode := continuous_mode;
	END_IF
UNTIL
	_executor = 0
END_REPEAT
END_SET
END_PROPERTY

METHOD create_container : I_Job
VAR_INPUT
	container_type	: ContainerType;
	name	: STRING;
END_VAR
CASE container_type OF
	ContainerType.BATCH:
		create_container := THIS^.create_job(GVL.batch_job_container_creator,name);
	ContainerType.PARALLEL:
		create_container := THIS^.create_job(GVL.parallel_job_container_creator,name);
	ContainerType.QUEUE:
		create_container := THIS^.create_job(GVL.queue_job_container_creator,name);
	ContainerType.PARALLEL_QUEUE:
		create_container := THIS^.create_job(GVL.parallel_queue_job_container_creator,name);
END_CASE
END_METHOD

METHOD create_job : I_Job
VAR_INPUT
	creator	: I_TaskCreator;
	future_name	: STRING;
END_VAR
VAR
	future : I_Future;
END_VAR
IF _num_of_jobs < ParamFuturesLib.MAX_TASK_NUM THEN
	future := creator.create_future(future_name);
	create_job := THIS^.spawn_job(future);
	create_job.persistent_job := FALSE;
	IF create_job <> 0 THEN
		create_job.future_creator := creator;
	ELSE
		creator.destroy_future(future);
	END_IF
END_IF
END_METHOD

PROPERTY each_executor : I_Job
GET
VAR
	_index : UINT;
END_VAR
_index := _index_generator_();
IF _index > 0 THEN
	IF _executors[_index] <> 0 THEN
		IF _executors[_index] <> 0 THEN
			each_executor := _executors[_index];
		ELSE
			each_executor := 0;
		END_IF
	END_IF
ELSE
	each_executor := 0;
END_IF
END_GET
END_PROPERTY

METHOD error_reset : BOOL
VAR
	_executor : I_Job;
	complete : BOOL;
END_VAR
complete := TRUE;
REPEAT
	_executor := each_executor;
	IF _executor <> 0 THEN
		IF NOT _executor.error_reset() THEN
			complete := FALSE;
		END_IF
	END_IF
UNTIL
	_executor = 0
END_REPEAT
IF complete THEN
	_error_id := 0;
END_IF
error_reset := complete;
END_METHOD

METHOD init : BOOL // Return TRUE if finish.
VAR
	_each_executor : i_Job;
	_init_done : BOOL;
END_VAR
_init_done := TRUE;
REPEAT
	_each_executor := THIS^.each_executor;
	IF _each_executor <> 0 THEN
		IF NOT _each_executor.init() THEN
			_init_done := FALSE;
		END_IF
	END_IF
UNTIL
	_each_executor = 0
END_REPEAT

_error_id := 0;
init := _init_done;
END_METHOD

PROPERTY num_of_jobs : UDINT
GET
num_of_jobs := _num_of_jobs;
END_GET
END_PROPERTY

METHOD reset : BOOL // Return TRUE if finish.
VAR_INPUT
	deep : BOOL := FALSE;
END_VAR
VAR
	i : UINT;
	_delete_counter : UINT;
	_p_executor : POINTER TO FB_Executor;
	text : STRING;
END_VAR
_delete_counter := 0;
REPEAT
	i := _index_generator_();
	IF _num_of_jobs > _delete_counter AND i > 0 THEN
		IF _executors[i] <> 0 THEN
			IF _executors[i].reset(deep) THEN
				IF __QUERYPOINTER(_executors[i],_p_executor) THEN
					__DELETE(_p_executor);
				ELSE
					_executors[i] := 0;
				END_IF
				_delete_counter := _delete_counter + 1;
			END_IF
		END_IF
	END_IF
UNTIL
	i = 0
END_REPEAT
_num_of_jobs := _num_of_jobs - _delete_counter;
reset := _num_of_jobs = 0;
END_METHOD

METHOD resume : BOOL
VAR
	_all_done : BOOL;
END_VAR
VAR_INST
	_executor : I_Job;
END_VAR
_all_done := TRUE;
REPEAT
	_executor := THIS^.each_executor;
	IF _executor <> 0 THEN
		IF NOT _executor.resume() THEN
			_all_done := FALSE;
		END_IF
	END_IF
UNTIL
	_executor = 0
END_REPEAT
resume := _all_done;
END_METHOD

METHOD spawn_job : I_Job
VAR_INPUT
	future : I_Future;
	job_persistence : BOOL := FALSE;
END_VAR
VAR
	_spawned_executor : POINTER TO FB_Executor;
END_VAR
IF future <> 0 THEN
	_spawned_executor := __NEW(FB_Executor);
	_spawned_executor^.future := future;
	_spawned_executor^.persistent_job := job_persistence;
	_append_job(_spawned_executor^);
	spawn_job := _spawned_executor^;
ELSE
	spawn_job := 0;
END_IF
END_METHOD

PROPERTY state : E_FutureExecutionState
GET
state := _state;
END_GET
SET
_state := state;
END_SET
END_PROPERTY

END_FUNCTION_BLOCK
